// TIA Portal project "FCs and FBs" (V15.1)

(* hardware
DEVICE "S71500/ET200MP station_1"  S7-1500 station
   slot 0: "Rail_0"  Rack  6ES7 590-1***0-0AA0
   slot 1: "PLC_1"  CPU 1516-3 PN/DP  6ES7 516-3AN01-0AB0  V2.6
      slot 3: "CPU display_1"  6ES7591-1BA00-0AA0
*)

// ===== PLC "PLC_1"  CPU 1516-3 PN/DP =====

VAR_GLOBAL   // PLC tag table "Default tag table"
   "Tag_1" AT %I0.0 : Bool;
   "Tag_2" AT %I0.1 : Bool;
   "Output Code" AT %QW10 : Int;
   "Up" AT %I1.0 : Bool;
   "Down" AT %I1.0 : Bool;
   "Infrared Code" AT %QW0 : Int;
   "V+" AT %I2.0 : Bool;
   "V-" AT %I2.0 : Bool;
   "Go Louder" AT %QW2 : Int;
END_VAR

DATA_BLOCK "Unicorn_2"   // DB4
{ S7_Optimized_Access := 'TRUE' }
VERSION : 0.1
// stored: InstanceOfName Filling
"Filling"
BEGIN
END_DATA_BLOCK

// folder: Data

DATA_BLOCK "Glass_1"   // DB1
{ S7_Optimized_Access := 'TRUE' }
VERSION : 0.1
// stored: InstanceOfName Filling
"Filling"
BEGIN
END_DATA_BLOCK

DATA_BLOCK "Glass_2"   // DB2
{ S7_Optimized_Access := 'TRUE' }
VERSION : 0.1
// stored: InstanceOfName Filling
"Filling"
BEGIN
END_DATA_BLOCK

DATA_BLOCK "Unicorn"   // DB3
{ S7_Optimized_Access := 'TRUE' }
VERSION : 0.1
// stored: InstanceOfName Filling
"Filling"
BEGIN
END_DATA_BLOCK

// folder: (top level)

FUNCTION_BLOCK "Filling"   // FB1, LAD
{ S7_Optimized_Access := 'TRUE' }
VERSION : 0.1
   VAR_INPUT
      "Fill In" : Bool;
      "Take Out" : Bool;
      "Volume Up" : Bool;
      "Volume Down" : Bool;
   END_VAR
   VAR_OUTPUT
      "Liquid Level" : Int;
      "Volume Code" : Int;
   END_VAR
   VAR
      "Fill Level Static" : Int;
   END_VAR
BEGIN

REGION Network 1: Fill In
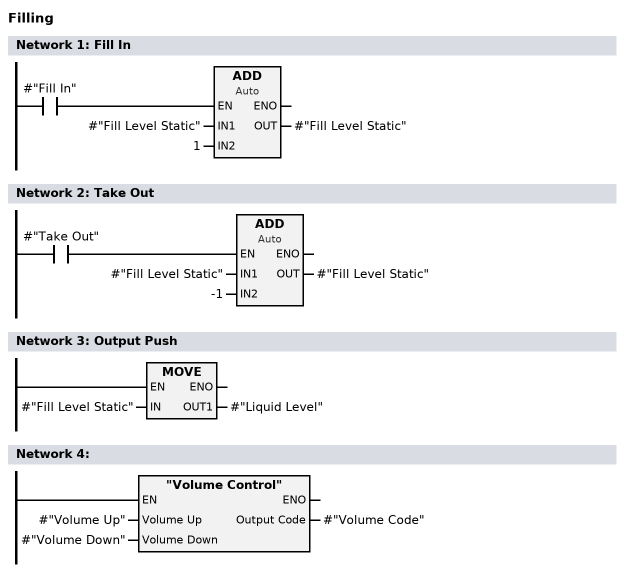
   RUNG wire#powerrail
      Contact( #"Fill In" )
      Add(in1 := #"Fill Level Static", in2 := 1, out => #"Fill Level Static")
   END_RUNG
   // the same network as SCL:
   IF #"Fill In" THEN #"Fill Level Static" := #"Fill Level Static" + 1; END_IF;
END_REGION

REGION Network 2: Take Out
   RUNG wire#powerrail
      Contact( #"Take Out" )
      Add(in1 := #"Fill Level Static", in2 := -1, out => #"Fill Level Static")
   END_RUNG
   // the same network as SCL:
   IF #"Take Out" THEN #"Fill Level Static" := #"Fill Level Static" + (-1); END_IF;
END_REGION

REGION Network 3: Output Push
   RUNG wire#powerrail
      Move(in := #"Fill Level Static", out1 => #"Liquid Level")
   END_RUNG
   // the same network as SCL:
   #"Liquid Level" := #"Fill Level Static";
END_REGION

REGION Network 4
   RUNG wire#powerrail
      "Volume Control"("Volume Up" := #"Volume Up", "Volume Down" := #"Volume Down", "Output Code" => #"Volume Code")
   END_RUNG
   // the same network as SCL:
   "Volume Control"("Volume Up" := #"Volume Up",
                    "Volume Down" := #"Volume Down",
                    "Output Code" => #"Volume Code");
END_REGION
END_FUNCTION_BLOCK

FUNCTION "Volume Control" : Void   // FC1, LAD
{ S7_Optimized_Access := 'TRUE' }
VERSION : 0.1
   VAR_INPUT
      "Volume Up" : Bool;
      "Volume Down" : Bool;
   END_VAR
   VAR_OUTPUT
      "Output Code" : Int;
   END_VAR
   VAR_TEMP
      "Output Code calc" : Int;
   END_VAR
   VAR CONSTANT
      "Code for Up" : Int := 30;
      "Code for Down" : Int := 31;
   END_VAR
BEGIN

REGION Network 1: Volume up
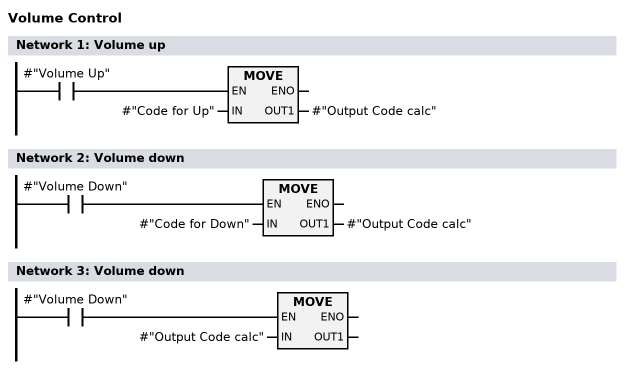
   RUNG wire#powerrail
      Contact( #"Volume Up" )
      Move(in := #"Code for Up", out1 => #"Output Code calc")
   END_RUNG
   // the same network as SCL:
   IF #"Volume Up" THEN #"Output Code calc" := #"Code for Up"; END_IF;
END_REGION

REGION Network 2: Volume down
   RUNG wire#powerrail
      Contact( #"Volume Down" )
      Move(in := #"Code for Down", out1 => #"Output Code calc")
   END_RUNG
   // the same network as SCL:
   IF #"Volume Down" THEN #"Output Code calc" := #"Code for Down"; END_IF;
END_REGION

REGION Network 3: Volume down
   RUNG wire#powerrail
      Contact( #"Volume Down" )
      Move(in := #"Output Code calc", out1 =>)
   END_RUNG
   // the same network as SCL:
   IF #"Volume Down" THEN <??.?> := #"Output Code calc"; END_IF;
END_REGION
END_FUNCTION

ORGANIZATION_BLOCK "Main"   // OB1, LAD, ProgramCycle
TITLE = "Main Program Sweep (Cycle)"
{ S7_Optimized_Access := 'TRUE' }
VERSION : 0.1
   VAR_INPUT
      Initial_Call : Bool;   // Initial call of this OB
      Remanence : Bool;   // =True, if remanent data are available
   END_VAR
BEGIN

REGION Network 1: Volume Control Call Remote 1
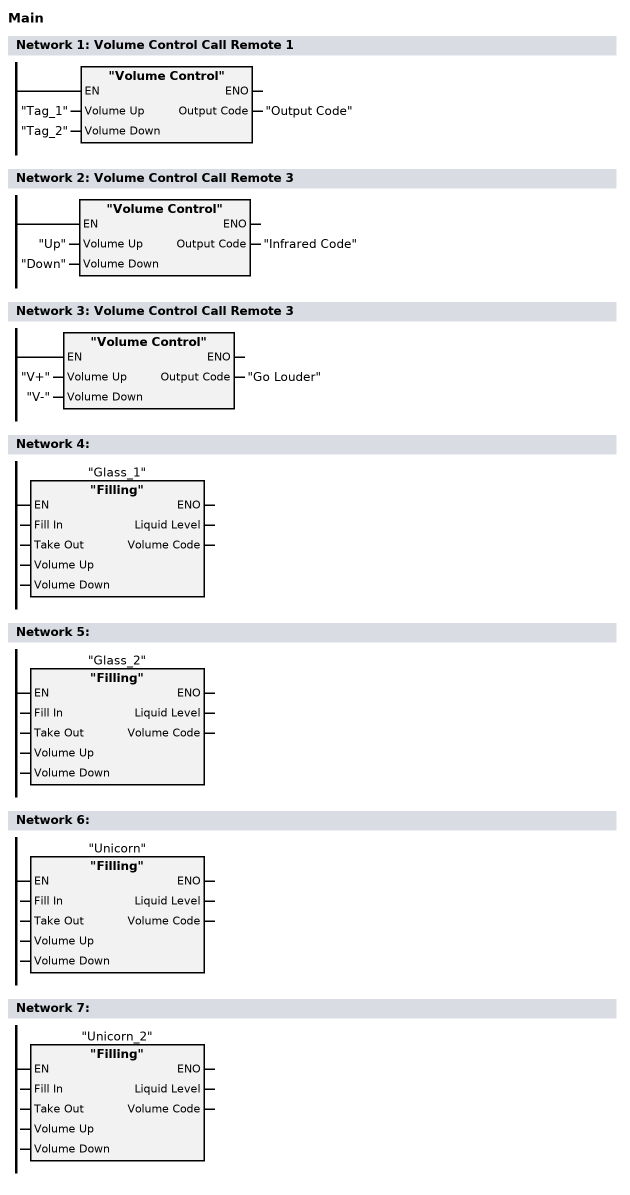
   RUNG wire#powerrail
      "Volume Control"("Volume Up" := "Tag_1", "Volume Down" := "Tag_2", "Output Code" => "Output Code")
   END_RUNG
   // the same network as SCL:
   "Volume Control"("Volume Up" := "Tag_1", "Volume Down" := "Tag_2", "Output Code" => "Output Code");
END_REGION

REGION Network 2: Volume Control Call Remote 3
   RUNG wire#powerrail
      "Volume Control"("Volume Up" := "Up", "Volume Down" := "Down", "Output Code" => "Infrared Code")
   END_RUNG
   // the same network as SCL:
   "Volume Control"("Volume Up" := "Up", "Volume Down" := "Down", "Output Code" => "Infrared Code");
END_REGION

REGION Network 3: Volume Control Call Remote 3
   RUNG wire#powerrail
      "Volume Control"("Volume Up" := "V+", "Volume Down" := "V-", "Output Code" => "Go Louder")
   END_RUNG
   // the same network as SCL:
   "Volume Control"("Volume Up" := "V+", "Volume Down" := "V-", "Output Code" => "Go Louder");
END_REGION

REGION Network 4
   RUNG wire#powerrail
      "Glass_1"("Fill In" :=, "Take Out" :=, "Volume Up" :=, "Volume Down" :=, "Liquid Level" =>, "Volume Code" =>)
   END_RUNG
   // the same network as SCL:
   "Glass_1"();   // "Filling"
END_REGION

REGION Network 5
   RUNG wire#powerrail
      "Glass_2"("Fill In" :=, "Take Out" :=, "Volume Up" :=, "Volume Down" :=, "Liquid Level" =>, "Volume Code" =>)
   END_RUNG
   // the same network as SCL:
   "Glass_2"();   // "Filling"
END_REGION

REGION Network 6
   RUNG wire#powerrail
      "Unicorn"("Fill In" :=, "Take Out" :=, "Volume Up" :=, "Volume Down" :=, "Liquid Level" =>, "Volume Code" =>)
   END_RUNG
   // the same network as SCL:
   "Unicorn"();   // "Filling"
END_REGION

REGION Network 7
   RUNG wire#powerrail
      "Unicorn_2"("Fill In" :=, "Take Out" :=, "Volume Up" :=, "Volume Down" :=, "Liquid Level" =>, "Volume Code" =>)
   END_RUNG
   // the same network as SCL:
   "Unicorn_2"();   // "Filling"
END_REGION
END_ORGANIZATION_BLOCK